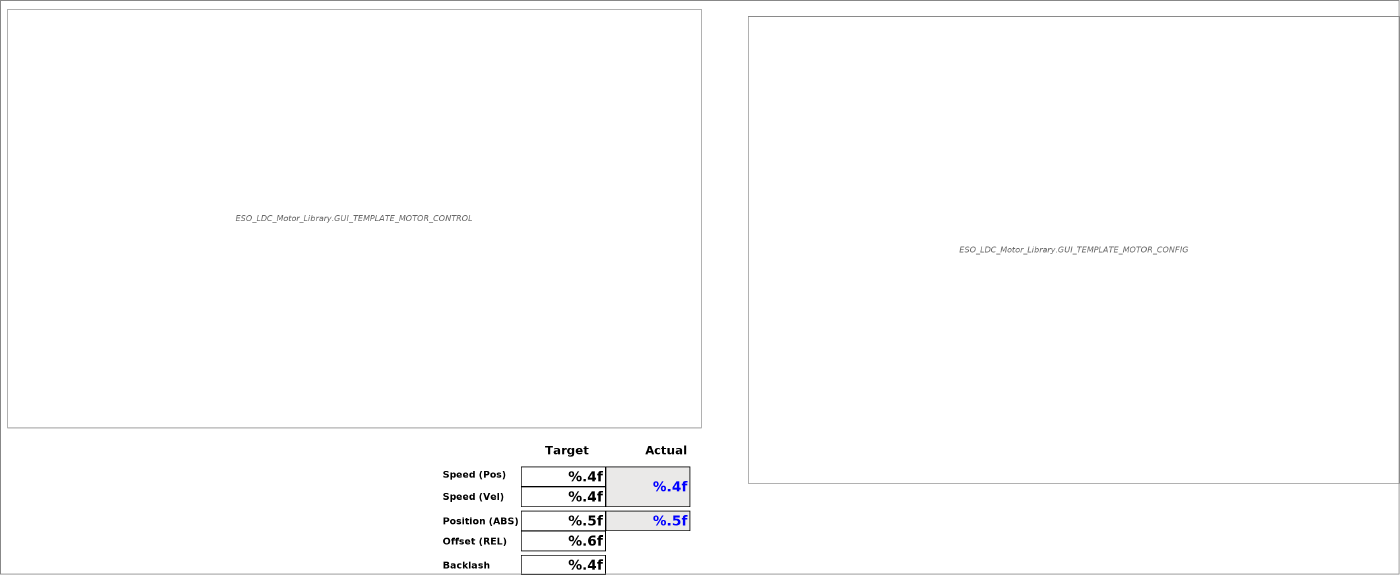
VISUALIZATION TipTilt_Servo_1  // 1739x715
    Frame (9,11 862x521)
        shows ESO_LDC_Motor_Library.GUI_TEMPLATE_MOTOR_CONTROL(m_Instance := MAIN.tiptilt_1)
    Frame (929,20 810x581)
        shows ESO_LDC_Motor_Library.GUI_TEMPLATE_MOTOR_CONFIG(m_Instance := MAIN.tiptilt_1)
    Rectangle (547,580 95x20), "Speed (Pos)"
    Rectangle (752,635 105x25), "%.5f", text variable: MAIN.tiptilt_1.stat.lrPosActual, input disabled if: false
    Rectangle (674,550 190x20), "Target Actual"
    Rectangle (547,638 95x20), "Position (ABS)"
    Rectangle (752,580 105x50), "%.4f", text variable: MAIN.tiptilt_1.stat.lrVelActual, input disabled if: false
    Rectangle (647,605 105x25), "%.4f", text variable: MAIN.tiptilt_1.ctrl.lrVelocity
        OnMouseDown: write the text variable via Default
    Rectangle (547,693 95x20), "Backlash"
    Rectangle (647,690 105x25), "%.4f", text variable: MAIN.tiptilt_1.cfg.lrBacklash
        OnMouseDown: write the text variable via Default
    Rectangle (547,605 95x25), "Speed (Vel)"
    Rectangle (647,635 105x25), "%.5f", tooltip "Absolute position used by "MOVE ABS"", text variable: MAIN.tiptilt_1.ctrl.lrPosition
        OnMouseDown: write the text variable via Default
    Rectangle (647,580 105x25), "%.4f", text variable: MAIN.tiptilt_1.cfg.lrDefaultVelocity
        OnMouseDown: write the text variable via Default
    Rectangle (547,663 95x20), "Offset (REL)"
    Rectangle (647,660 105x25), "%.6f", tooltip "Relative offset used by "MOVE REL"", text variable: MAIN.tiptilt_1.ctrl.lrOffset
        OnMouseDown: write the text variable via Default
END_VISUALIZATION

(* stored: Version 1.1.0.1, ProductVersion 3.1.4024.12
   Visu TipTilt_Servo_1: Id {8e9a6828-5b88-4d1c-ad60-7f2a825e9e85} *)
